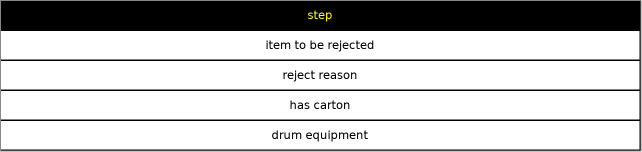
VISUALIZATION CARTON_PICKUP_SHIFT_ELEMENT_DESCRIPTION  // 642x152
    Rectangle (0,0 640x30), "step"
    Rectangle (0,30 640x30), "item to be rejected"
    Rectangle (0,60 640x30), "reject reason"
    Rectangle (0,90 640x30), "has carton"
    Rectangle (0,120 640x30), "drum equipment"
END_VISUALIZATION

(* stored: Version 1.1.0.1, ProductVersion 3.1.4024.3
   Visu CARTON_PICKUP_SHIFT_ELEMENT_DESCRIPTION: Id {c965c0c0-5229-46ec-951e-1955596eb30a} *)
